FUNCTION_BLOCK INI_AR2IO (* Load and Store REAL Data from settings.ini by Section and Key (AR Adapter Interface) *)
  (* Standard: 61499-2; Description: Copyright (c) 2026 Meisterschulen am Ostbahnhof This program and the accompanying materials are made available under the terms of the Eclipse Public License 2.0 which is available at https://www.eclipse.org/legal/epl-2.0/ SPDX-License-Identifier: EPL-2.0 *)
  (* Version 1.0, 2026-04-24, Franz Höpfinger, Meisterschulen am Ostbahnhof, initial API and implementation and/or initial documentation *)
  PACKAGE logiBUS::storage::ini;
  IMPORT eclipse4diac::core::TypeHash;
  IMPORT adapter::types::unidirectional::AR;
  IMPORT eclipse4diac::storage::INI;
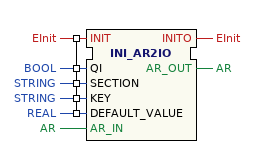
  EVENT_INPUT
    INIT : EInit WITH QI, SECTION, KEY, DEFAULT_VALUE; (* Service Initialization *)
  END_EVENT
  EVENT_OUTPUT
    INITO : EInit; (* Initialization Confirm *)
  END_EVENT
  VAR_INPUT
    QI : BOOL; (* Event Input Qualifier *)
    SECTION : STRING; (* Section name. *)
    KEY : STRING; (* Key name. *)
    DEFAULT_VALUE : REAL; (* The value to read if there is nothing in the settings.ini *)
  END_VAR
  SOCKETS
    AR_IN : adapter::types::unidirectional::AR; (* Value to store (SET) *)
  END_SOCKETS
  PLUGS
    AR_OUT : adapter::types::unidirectional::AR; (* Stored value output (GETO) *)
  END_PLUGS
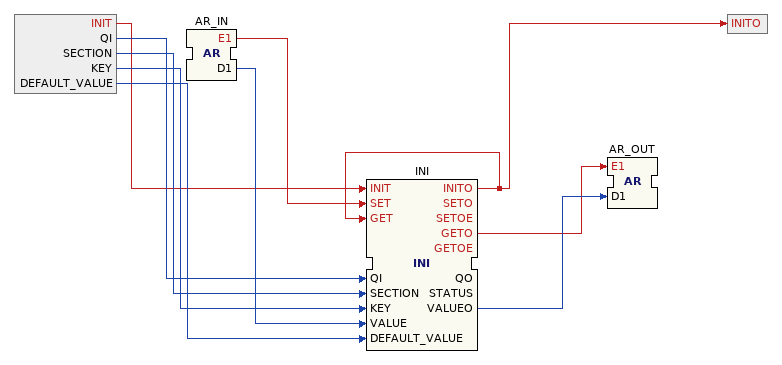
  FBS
    INI : eclipse4diac::storage::INI;
  END_FBS
  EVENT_CONNECTIONS
    INIT TO INI.INIT;
    INI.INITO TO INITO;
    INI.INITO TO INI.GET;
    AR_IN.E1 TO INI.SET;
    INI.GETO TO AR_OUT.E1;
  END_CONNECTIONS
  DATA_CONNECTIONS
    QI TO INI.QI;
    SECTION TO INI.SECTION;
    KEY TO INI.KEY;
    DEFAULT_VALUE TO INI.DEFAULT_VALUE;
    AR_IN.D1 TO INI.VALUE;
    INI.VALUEO TO AR_OUT.D1;
  END_CONNECTIONS
END_FUNCTION_BLOCK
